TYPE ST_Inverter_Write :
STRUCT
	Controlword				: ST_InverterControlWord;
	ui_ControlwordValue		: UINT;
	i_invertermode 			: INT;
	i_BaseCurrentRef 		: INT;
	i_ReactiveCurrentRef	: INT;
	i_FrequencyDroop		: INT;
	i_VoltageDroop			: INT;
	i_FrequencyDroopOffset	: INT;
	i_VoltageCorrection		: INT;
	i_BaseRefRampRate		: INT;
	i_StartPowerMode		: INT;
	i_StartVoltageMode		: INT;
	i_OutActCurrentLimit	: INT;
	i_InActCurrentLimit		: INT;
	i_DCVramprate			: INT;
END_STRUCT
END_TYPE

(* stored: Version 1.1.0.1, ProductVersion 3.1.4026.18
   DUT ST_Inverter_Write: Id {489ace50-f893-4b6f-8465-2e940359943b} *)
